// TIA Portal V17 export
// export: Created 2025-03-10T13:10:09.7625003Z, ExportSetting WithDefaults, DisplayName Totally Integrated Automation Portal, DisplayVersion V17 Update 8, DisplayName TIA Portal Openness, DisplayVersion V17 Update 8, DisplayName TIA Portal Version Control Interface, DisplayVersion V17, DisplayName SINAMICS Startdrive Advanced, DisplayVersion V17 SP2, DisplayName SINAMICS Startdrive G110M, G120, G120C, G120D, G120P, G115D, DisplayVersion V17 SP2, DisplayName SINAMICS Startdrive G130, G150, S120, S150, SINAMICS MV, S210, DisplayVersion V17 SP2, DisplayName STEP 7 Professional, DisplayVersion V17 Update 8, DisplayName SINUMERIK ONE STEP 7 Toolbox, DisplayVersion V17 Update 12, DisplayName SINUMERIK 840D sl STEP 7 Toolbox, DisplayVersion V17 Update 12, DisplayName STEP 7 Safety, DisplayVersion V17 Update 6, DisplayName WinCC Advanced, DisplayVersion V17 Update 8
DATA_BLOCK "DB307_CH7_READ_AXES_POSITIONS"   // DB307
{ DB_Accessible_From_OPC_UA := 'FALSE' }
AUTHOR : ETXETAR
VERSION : 1.0
// stored: AutoNumber false, DBAccessibleFromOPCUA false, DBAccessibleFromWebserver true, InstanceOfName FB301_CHANNEL_READ_AXES_POSITIONS, InstanceOfType FB
"FB301_CHANNEL_READ_AXES_POSITIONS"
   // VAR_INPUT
   //    NUMBER_AXES_GROUP_1 : Int;
   //    NUMBER_AXES_GROUP_2 : Int;
   //    NUMBER_AXES_GROUP_3 : Int;
   // END_VAR
   // VAR_OUTPUT
   //    ALARM : Bool;
   //    AXIS_POSITION_1 : DWord;
   //    AXIS_POSITION_2 : DWord;
   //    AXIS_POSITION_3 : DWord;
   //    AXIS_POSITION_4 : DWord;
   //    AXIS_POSITION_5 : DWord;
   //    AXIS_POSITION_6 : DWord;
   //    AXIS_POSITION_7 : DWord;
   //    AXIS_POSITION_8 : DWord;
   //    AXIS_POSITION_9 : DWord;
   //    AXIS_POSITION_10 : DWord;
   //    AXIS_POSITION_11 : DWord;
   //    AXIS_POSITION_12 : DWord;
   //    AXIS_POSITION_13 : DWord;
   //    AXIS_POSITION_14 : DWord;
   //    AXIS_POSITION_15 : DWord;
   //    AXIS_POSITION_16 : DWord;
   //    AXIS_POSITION_17 : DWord;
   //    AXIS_POSITION_18 : DWord;
   //    AXIS_POSITION_19 : DWord;
   //    AXIS_POSITION_20 : DWord;
   // END_VAR
   // VAR RETAIN
   //    readDB { S7_SetPoint := 'True'} : "READ_AXES_POSITIONS_CH";
   //    FB2_Instance_1 { S7_SetPoint := 'True'} : "LBP_ReadVar";
   //    FB2_Instance_2 { S7_SetPoint := 'True'} : "LBP_ReadVar";
   //    FB2_Instance_3 { S7_SetPoint := 'True'} : "LBP_ReadVar";
   //    FAULT_COUNTER { S7_SetPoint := 'True'} : CTU_INT;
   // END_VAR
BEGIN
   readDB.CH_Reading_1.Area_Unit := BYTE#16#47;
   readDB.CH_Reading_2.Area_Unit := BYTE#16#47;
   readDB.CH_Reading_3.Area_Unit := BYTE#16#47;
   readDB.CH_Reading_4.Area_Unit := BYTE#16#47;
   readDB.CH_Reading_5.Area_Unit := BYTE#16#47;
   readDB.CH_Reading_6.Area_Unit := BYTE#16#47;
   readDB.CH_Reading_7.Area_Unit := BYTE#16#47;
   readDB.CH_Reading_8.Area_Unit := BYTE#16#47;
   readDB.CH_Reading_9.Area_Unit := BYTE#16#47;
   readDB.CH_Reading_10.Area_Unit := BYTE#16#47;
   readDB.CH_Reading_11.Area_Unit := BYTE#16#47;
   readDB.CH_Reading_12.Area_Unit := BYTE#16#47;
   readDB.CH_Reading_13.Area_Unit := BYTE#16#47;
   readDB.CH_Reading_14.Area_Unit := BYTE#16#47;
   readDB.CH_Reading_15.Area_Unit := BYTE#16#47;
   readDB.CH_Reading_16.Area_Unit := BYTE#16#47;
   readDB.CH_Reading_17.Area_Unit := BYTE#16#47;
   readDB.CH_Reading_18.Area_Unit := BYTE#16#47;
   readDB.CH_Reading_19.Area_Unit := BYTE#16#47;
   readDB.CH_Reading_20.Area_Unit := BYTE#16#47;
END_DATA_BLOCK
